// TIA Portal V19 export
TYPE "C701_STU_IF_KMI_TYPIC"
   STRUCT
      CMD_NORM { ExternalAccessible := 'False'; ExternalVisible := 'False'; ExternalWritable := 'False'} : Bool;   // Aansturing klimaatregeling in stand Normaal (1 = Aan)
      CMD_CIR { ExternalAccessible := 'False'; ExternalVisible := 'False'; ExternalWritable := 'False'} : Bool;   // Aansturing klimaatregeling in stand Recirculatie (1 = Aan)
   END_STRUCT;
END_TYPE
